{attribute 'linkalways'} 
{attribute 'no_explicit_call' := 'This FB is a CLASS and must be accessed using methods or properties'}
{attribute 'enable_dynamic_creation'}
FUNCTION_BLOCK _REAL EXTENDS NumericDatatypeBase
VAR
	localData : REAL;
	activeData : REFERENCE TO REAL REF= localData;
END_VAR

PROPERTY PUBLIC Address : PVOID
GET
Address := ADR(activeData);
END_GET
END_PROPERTY

METHOD PUBLIC ClearReference
VAR_INPUT
END_VAR
activeData REF= localData;
END_METHOD

METHOD PUBLIC Clone : I_Datatype
VAR
    pClone : POINTER TO _REAL;
END_VAR
pClone := __NEW(_REAL(InitialValue := Value));
Clone := pClone^;
END_METHOD

METHOD FB_init : BOOL
VAR_INPUT
	bInitRetains : BOOL; // if TRUE, the retain variables are initialized (warm start / cold start)
	bInCopyCode : BOOL;  // if TRUE, the instance afterwards gets moved into the copy code (online change)
	InitialValue : REAL;
END_VAR
localData := InitialValue;
END_METHOD

PROPERTY PUBLIC IsFloat : BOOL
GET
IsFloat := TRUE;
END_GET
END_PROPERTY

PROPERTY PUBLIC IsSigned : BOOL
GET
IsSigned := TRUE;
END_GET
END_PROPERTY

METHOD PUBLIC MakeReferenceTo
VAR_INPUT
	ReferenceTarget : REFERENCE TO REAL;
END_VAR
activeData REF= ReferenceTarget;
END_METHOD

PROPERTY PUBLIC MaxValue : REAL
GET
MaxValue :=  DatatypeLimits.REAL_MAX_VALUE;
END_GET
END_PROPERTY

PROPERTY PUBLIC MinValue : REAL
GET
MinValue := DatatypeLimits.REAL_MIN_VALUE;
END_GET
END_PROPERTY

METHOD PROTECTED SerializeMaxValue
VAR_INPUT
	Serializer : I_Serializer;
END_VAR
Serializer.AddReal(MaxValue);
END_METHOD

METHOD PROTECTED SerializeMinValue
VAR_INPUT
	Serializer : I_Serializer;
END_VAR
Serializer.AddReal(MinValue);
END_METHOD

METHOD PUBLIC SerializeWith
VAR_INPUT
	Serializer : I_Serializer;
END_VAR
Serializer.AddReal(activeData);
END_METHOD

PROPERTY PUBLIC Size : UDINT
GET
Size := SIZEOF(activeData);
END_GET
END_PROPERTY

METHOD TryDeserializeFrom : BOOL
VAR_INPUT
	Deserializer : I_Deserializer;
	Feedback : I_DeserializerFeedback;
END_VAR
TryDeserializeFrom := Deserializer.TryGetReal(activeData, Feedback);
END_METHOD

METHOD TryMakeReferenceTo : BOOL
VAR_INPUT
	Target : I_Datatype;
END_VAR
VAR
	pTargetData : POINTER TO REAL;
END_VAR
IF NOT (Target.TypeName = TypeName) THEN
	RETURN;
END_IF

pTargetData := Target.Address;
activeData REF= pTargetData^;
TryMakeReferenceTo := TRUE;
END_METHOD

PROPERTY PUBLIC TypeName : T_MAXSTRING
GET
TypeName := 'REAL';
END_GET
END_PROPERTY

PROPERTY PUBLIC Value : REAL
GET
Value := activeData;
END_GET
SET
activeData := Value;
END_SET
END_PROPERTY

END_FUNCTION_BLOCK

(* stored: Version 1.1.0.1, ProductVersion 3.1.4024.12
   POU _REAL: Id {0705be22-a7a9-47ef-8afc-cf0c036d2b5e}, SpecialFunc None
   Folder Constructor: Id {dfaff8b4-7148-476b-9226-dc57d57bf216}
   Folder Protected: Id {db23cea0-72e4-0219-3f37-c7272deb623f}
   Property Address: Id {3e47a9d6-f9d2-4b84-9ed1-0be93fed72ea}
   Get Get: Id {ddc89f16-4171-4f6b-85e5-bcf033872e70}
   Method ClearReference: Id {f2d7e3d0-d7ec-47d2-9492-303b2dba55c7}
   Method Clone: Id {382ad76a-6a8f-423f-968d-5178e6ae96c4}
   Method FB_init: Id {b86268bf-faf6-452c-92ad-2861bd490861}
   Property IsFloat: Id {310f057c-dbcb-4b07-ba31-ce8872e27581}
   Get Get: Id {169db661-3d45-46d6-8f2d-2a55d675edbc}
   Property IsSigned: Id {936273a5-8441-4302-81dd-9a2c3290c284}
   Get Get: Id {3fc180d3-86bb-40dc-9d24-6b008e4c5175}
   Method MakeReferenceTo: Id {8c7b97e9-066e-436e-b653-da0c953a25bc}
   Property MaxValue: Id {9f3033b9-f4b2-05a7-3822-c7777f507e94}
   Get Get: Id {a3242c94-f95a-0637-1cbd-9cbd0419ba9d}
   Property MinValue: Id {95824644-e30e-0cd3-2ebf-8da96b38d866}
   Get Get: Id {004c8db9-92d7-07ba-2221-cec18ecfc3a8}
   Method SerializeMaxValue: Id {c9a429d4-5f3b-0bfb-0b12-24705981015b}
   Method SerializeMinValue: Id {6d2c181e-3e5c-0f2c-377d-54dbd4158eec}
   Method SerializeWith: Id {b0100a82-b2e0-4edd-b232-a90cec9f2427}
   Property Size: Id {cd91d3ef-1bbd-400e-a78f-952e2616e768}
   Get Get: Id {2695954d-6ede-4963-a006-def649e6b043}
   Method TryDeserializeFrom: Id {83c7d43d-b513-406d-87e3-eca6b0848a0c}
   Method TryMakeReferenceTo: Id {dd97e46d-1f2c-415a-94e1-0f4983bb4699}
   Property TypeName: Id {2ba520ec-dd25-4eab-974a-fc7af6a1ee2b}
   Get Get: Id {ff09c425-01e2-4b18-bd76-2d428a67685a}
   Property Value: Id {0a40f8eb-1bbe-4a00-afe1-c1b3b1f158c0}
   Get Get: Id {72b163f4-3cbd-4d9f-b627-4ccd7b588465}
   Set Set: Id {12860781-2c65-46ab-88d0-45040884c998} *)
